REGION Network 121: [Ax] - Manipolatori Testa/Coda - RIFERIMENTI
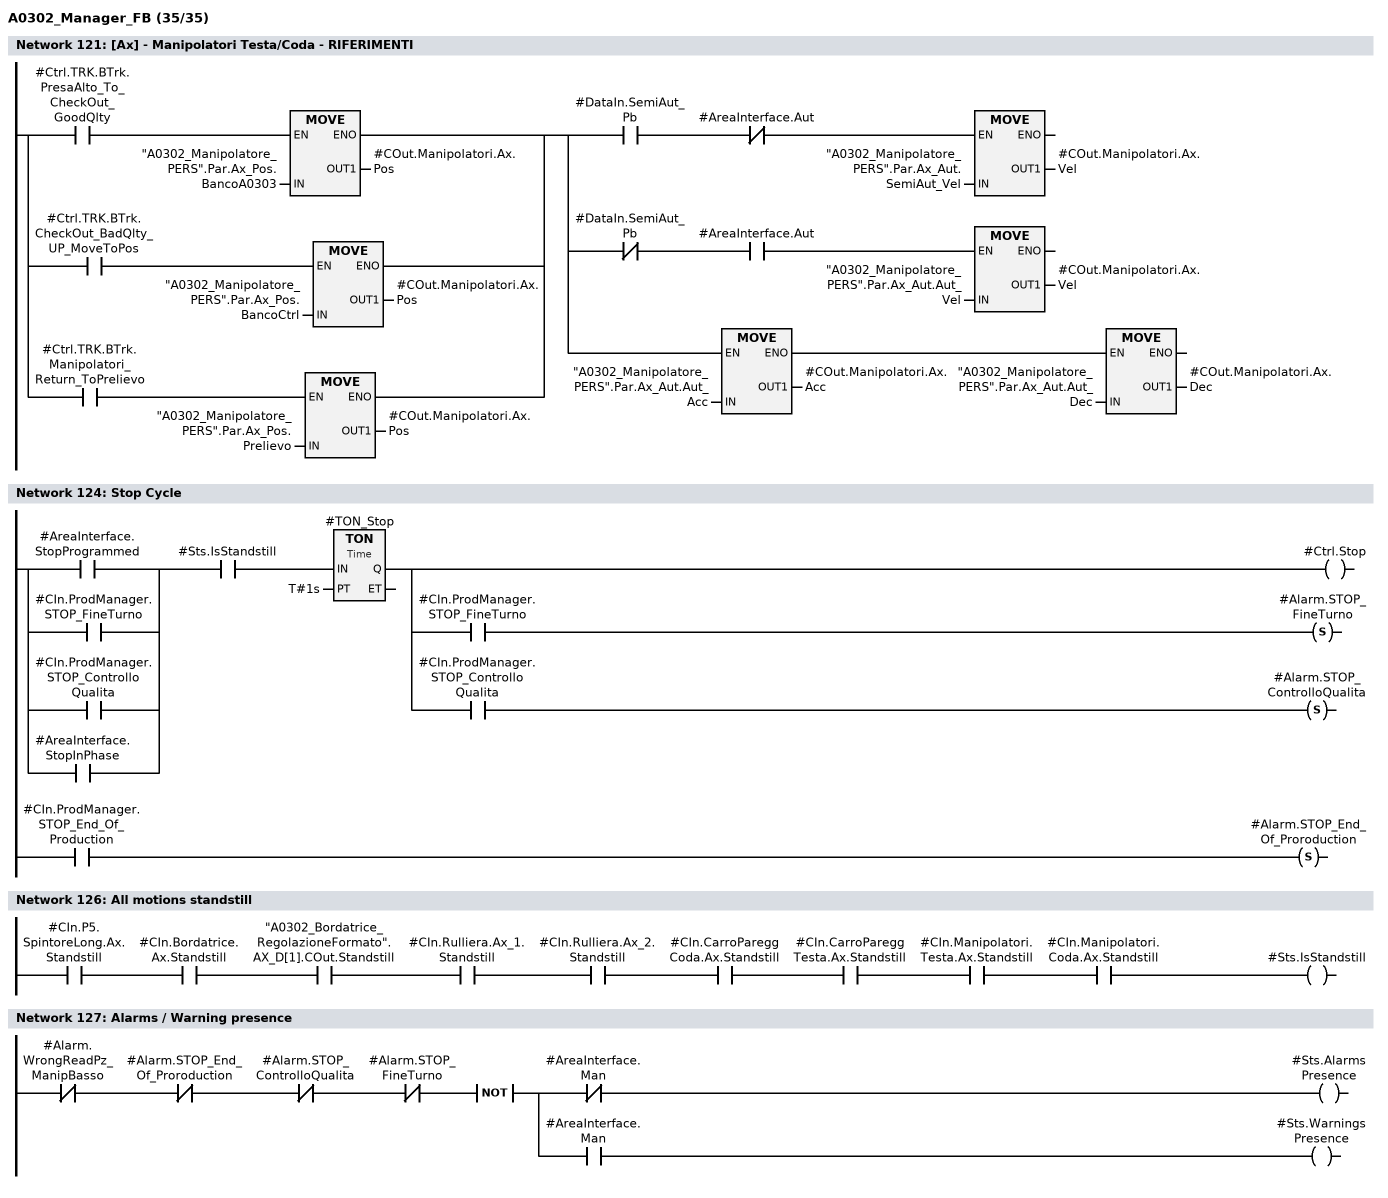
   RUNG wire#powerrail
      Contact( #Ctrl.TRK.BTrk.PresaAlto_To_CheckOut_GoodQlty )
      Move(in := "A0302_Manipolatore_PERS".Par.Ax_Pos.BancoA0303, out1 => #COut.Manipolatori.Ax.Pos)
      wire#w1
      Contact( #DataIn.SemiAut_Pb )
      I_Contact( #AreaInterface.Aut )
      Move(in := "A0302_Manipolatore_PERS".Par.Ax_Aut.SemiAut_Vel, out1 => #COut.Manipolatori.Ax.Vel)
   END_RUNG
   RUNG wire#powerrail
      Contact( #Ctrl.TRK.BTrk.CheckOut_BadQlty_UP_MoveToPos )
      Move(in := "A0302_Manipolatore_PERS".Par.Ax_Pos.BancoCtrl, out1 => #COut.Manipolatori.Ax.Pos)
   END_RUNG wire#w1
   RUNG wire#powerrail
      Contact( #Ctrl.TRK.BTrk.Manipolatori_Return_ToPrelievo )
      Move(in := "A0302_Manipolatore_PERS".Par.Ax_Pos.Prelievo, out1 => #COut.Manipolatori.Ax.Pos)
   END_RUNG wire#w1
   RUNG wire#w1
      I_Contact( #DataIn.SemiAut_Pb )
      Contact( #AreaInterface.Aut )
      Move(in := "A0302_Manipolatore_PERS".Par.Ax_Aut.Aut_Vel, out1 => #COut.Manipolatori.Ax.Vel)
   END_RUNG
   RUNG wire#w1
      Move(in := "A0302_Manipolatore_PERS".Par.Ax_Aut.Aut_Acc, out1 => #COut.Manipolatori.Ax.Acc)
      Move(in := "A0302_Manipolatore_PERS".Par.Ax_Aut.Aut_Dec, out1 => #COut.Manipolatori.Ax.Dec)
   END_RUNG
   // the same network as SCL:
   IF #Ctrl.TRK.BTrk.PresaAlto_To_CheckOut_GoodQlty THEN
       #COut.Manipolatori.Ax.Pos := "A0302_Manipolatore_PERS".Par.Ax_Pos.BancoA0303;
   END_IF;
   IF #Ctrl.TRK.BTrk.CheckOut_BadQlty_UP_MoveToPos THEN
       #COut.Manipolatori.Ax.Pos := "A0302_Manipolatore_PERS".Par.Ax_Pos.BancoCtrl;
   END_IF;
   IF #Ctrl.TRK.BTrk.Manipolatori_Return_ToPrelievo THEN
       #COut.Manipolatori.Ax.Pos := "A0302_Manipolatore_PERS".Par.Ax_Pos.Prelievo;
   END_IF;
   #_w1 := #Ctrl.TRK.BTrk.PresaAlto_To_CheckOut_GoodQlty OR #Ctrl.TRK.BTrk.CheckOut_BadQlty_UP_MoveToPos OR #Ctrl.TRK.BTrk.Manipolatori_Return_ToPrelievo;
   IF #_w1 AND #DataIn.SemiAut_Pb AND NOT #AreaInterface.Aut THEN
       #COut.Manipolatori.Ax.Vel := "A0302_Manipolatore_PERS".Par.Ax_Aut.SemiAut_Vel;
   END_IF;
   IF #_w1 AND NOT #DataIn.SemiAut_Pb AND #AreaInterface.Aut THEN
       #COut.Manipolatori.Ax.Vel := "A0302_Manipolatore_PERS".Par.Ax_Aut.Aut_Vel;
   END_IF;
   IF #_w1 THEN
       #COut.Manipolatori.Ax.Acc := "A0302_Manipolatore_PERS".Par.Ax_Aut.Aut_Acc;
       #COut.Manipolatori.Ax.Dec := "A0302_Manipolatore_PERS".Par.Ax_Aut.Aut_Dec;
   END_IF;
END_REGION

REGION Network 122: <+>
END_REGION

REGION Network 124: Stop Cycle
   RUNG wire#powerrail
      Contact( #AreaInterface.StopProgrammed )
      wire#w1
      Contact( #Sts.IsStandstill )
      { S7_Templates := "time_type := Time" } #TON_Stop.TON(pt := T#1s, et =>)
      wire#w2
      Coil( #Ctrl.Stop )
   END_RUNG
   RUNG wire#powerrail
      Contact( #CIn.ProdManager.STOP_FineTurno )
   END_RUNG wire#w1
   RUNG wire#powerrail
      Contact( #CIn.ProdManager.STOP_ControlloQualita )
   END_RUNG wire#w1
   RUNG wire#powerrail
      Contact( #AreaInterface.StopInPhase )
   END_RUNG wire#w1
   RUNG wire#w2
      Contact( #CIn.ProdManager.STOP_FineTurno )
      S_Coil( #Alarm.STOP_FineTurno )
   END_RUNG
   RUNG wire#w2
      Contact( #CIn.ProdManager.STOP_ControlloQualita )
      S_Coil( #Alarm.STOP_ControlloQualita )
   END_RUNG
   RUNG wire#powerrail
      Contact( #CIn.ProdManager.STOP_End_Of_Production )
      S_Coil( #Alarm.STOP_End_Of_Proroduction )
   END_RUNG
   // the same network as SCL:
   #TON_Stop.TON(IN := (#AreaInterface.StopProgrammed OR #CIn.ProdManager.STOP_FineTurno OR #CIn.ProdManager.STOP_ControlloQualita OR #AreaInterface.StopInPhase) AND #Sts.IsStandstill,
                 PT := T#1s);
   #Ctrl.Stop := #TON_Stop.Q;
   IF #TON_Stop.Q AND #CIn.ProdManager.STOP_FineTurno THEN #Alarm.STOP_FineTurno := TRUE; END_IF;
   IF #TON_Stop.Q AND #CIn.ProdManager.STOP_ControlloQualita THEN
       #Alarm.STOP_ControlloQualita := TRUE;
   END_IF;
   IF #CIn.ProdManager.STOP_End_Of_Production THEN #Alarm.STOP_End_Of_Proroduction := TRUE; END_IF;
END_REGION

REGION Network 125: << FINAL OPERATIONS >>
   // +
   // +
   // +
   // +
   // +
   // +
   // +
   // +
   // +
   // +
   // +
   // +
   // +
END_REGION

REGION Network 126: All motions standstill
   RUNG wire#powerrail
      Contact( #CIn.P5.SpintoreLong.Ax.Standstill )
      Contact( #CIn.Bordatrice.Ax.Standstill )
      Contact( "A0302_Bordatrice_RegolazioneFormato".AX_D[1].COut.Standstill )
      Contact( #CIn.Rulliera.Ax_1.Standstill )
      Contact( #CIn.Rulliera.Ax_2.Standstill )
      Contact( #CIn.CarroPareggCoda.Ax.Standstill )
      Contact( #CIn.CarroPareggTesta.Ax.Standstill )
      Contact( #CIn.Manipolatori.Testa.Ax.Standstill )
      Contact( #CIn.Manipolatori.Coda.Ax.Standstill )
      Coil( #Sts.IsStandstill )
   END_RUNG
   // the same network as SCL:
   #Sts.IsStandstill := #CIn.P5.SpintoreLong.Ax.Standstill AND #CIn.Bordatrice.Ax.Standstill AND "A0302_Bordatrice_RegolazioneFormato".AX_D[1].COut.Standstill AND #CIn.Rulliera.Ax_1.Standstill AND #CIn.Rulliera.Ax_2.Standstill AND #CIn.CarroPareggCoda.Ax.Standstill AND #CIn.CarroPareggTesta.Ax.Standstill AND #CIn.Manipolatori.Testa.Ax.Standstill AND #CIn.Manipolatori.Coda.Ax.Standstill;
END_REGION

REGION Network 127: Alarms / Warning presence
   RUNG wire#powerrail
      I_Contact( #Alarm.WrongReadPz_ManipBasso )
      I_Contact( #Alarm.STOP_End_Of_Proroduction )
      I_Contact( #Alarm.STOP_ControlloQualita )
      I_Contact( #Alarm.STOP_FineTurno )
      Not()
      wire#w1
      I_Contact( #AreaInterface.Man )
      Coil( #Sts.AlarmsPresence )
   END_RUNG
   RUNG wire#w1
      Contact( #AreaInterface.Man )
      Coil( #Sts.WarningsPresence )
   END_RUNG
   // the same network as SCL:
   #_w1 := NOT (NOT #Alarm.WrongReadPz_ManipBasso AND NOT #Alarm.STOP_End_Of_Proroduction AND NOT #Alarm.STOP_ControlloQualita AND NOT #Alarm.STOP_FineTurno);
   #Sts.AlarmsPresence := #_w1 AND NOT #AreaInterface.Man;
   #Sts.WarningsPresence := #_w1 AND #AreaInterface.Man;
END_REGION

REGION Network 128 (SCL): Collect machine to area interface
   #MachineInterface.AlarmsPresence := #Sts.AlarmsPresence;

   #MachineInterface.WarningPresence := #Sts.WarningsPresence;

   #MachineInterface.MotionsStandStill := #Sts.IsStandstill;

   #MachineInterface.AutReady := #AreaInterface.Aut AND NOT #Sts.AlarmsPresence;


   #MachineInterface.AckStopInPhase := #AreaInterface.StopInPhase AND #Ctrl.Stop;

   #MachineInterface.AckStopProgrammed := #AreaInterface.StopProgrammed AND #Ctrl.Stop;


   #MachineInterface.Aborting := #AreaInterface.Aut AND #Sts.AlarmsPresence;
END_REGION
END_FUNCTION_BLOCK
